FUNCTION_BLOCK CONSOLE (* Console Output Service Interface *)
  (* Standard: 61499-1; Classification: Debugging; Function: Console I/O *)
  (* Version 0.0, 2003-03-26, JHC, Rockwell Automation *)
  (* Compiler header: package fb.rt; *)
  (* Compiler Java Sun javac(NetBeans) 1.4.1 *)
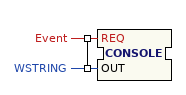
  EVENT_INPUT
    REQ WITH OUT;
  END_EVENT
  VAR_INPUT
    OUT : WSTRING; (* Data to write to console *)
  END_VAR
END_FUNCTION_BLOCK
